Fanuc KAREL source: test_csv_write.kl

PROGRAM test_csv_wrt
%NOLOCKGROUP

%include csv.klh

CONST
  PIPE_FILE = 'PIP:TESTCSV.DAT'
  CSV_FILE = 'FR:testcsv.csv'

VAR
  write_fl : FILE

BEGIN
END test_csv_wrt
